{attribute 'qualified_only'}
TYPE ENUM_TM2K2_States :
// Adapted from ENUM_ATM_States to add TARGET6
(
    Unknown := 0,
    OUT := 1,
    TARGET1 := 2,
    TARGET2 := 3,
    TARGET3 := 4,
    TARGET4 := 5,
    TARGET5 := 6,
    TARGET6 := 7
);
END_TYPE

(* stored: Version 1.1.0.1, ProductVersion 3.1.4022.18
   DUT ENUM_TM2K2_States: Id {39e72780-ebe1-47a1-93c3-70f8a4ded457} *)
